FUNCTION_BLOCK PUBLIC RejectStation
VAR_INPUT
END_VAR
VAR_OUTPUT
END_VAR
VAR
	xTrigger :BOOL := FALSE; // triggers processing
	State : eRejectStaState := eRejectStaState.eUnknown;
	NextState : eRejectStaState := eRejectStaState.eUnknown;
	ErrorReturnState : eRejectStaState := eRejectStaState.eUnknown;
	bFirst : BOOL := TRUE;
	VUT : BYTE; //VehicleID Under Station
	DwellTimer : TON;
	StateTimer : TON;
END_VAR

IF (GVL_IO.MachineEStopped) THEN 
	State := eRejectStaState.eUnknown;
	NextState := eRejectStaState.eUnknown;
	Status.RejectStatusMsg:= 'RejectSta Unknown, Check AIR, E-STOP and Hit Start';
END_IF

CASE State OF
eRejectStaState.eUnknown:
	Status.RejectStatusMsg:= 'RejectSta Unknown, Check AIR, E-STOP and Hit Start';
    IF (GVL_IO.MC_XStartPB AND GVL_IO.MC_XAirPressureOK AND GVL_IO.MC_NotEStopped) THEN // wait for start button when powered up or PLC program restarted
		NextState := eRejectStaState.eInit;	   
	END_IF
    

eRejectStaState.eInit:
    Act_KnockPartOFF();
	Act_FreePalletHoldDown();
	ResetDwellTimer();
	NextState := eRejectStaState.eHoming;
	

eRejectStaState.eHoming:
	IF (IsPalletHoldDownFree()) THEN 
         NextState := eRejectStaState.eReady;
	  END_IF
     DwellTimer(IN:=TRUE, PT:= T#10S);
     IF (DwellTimer.Q) THEN
		 ResetDwellTimer();
		 ErrorReturnState:= eRejectStaState.eInit;
		 NextState := eRejectStaState.eError;		 
	 END_IF	

eRejectStaState.eReady:
	IF (xTrigger) THEN
		NextState := eRejectStaState.eSendPalletHoldDownExtend;		
		ResetDwellTimer();
	END_IF

eRejectStaState.eSendPalletHoldDownExtend:
	Act_EngagePalletHoldDown();
	ResetDwellTimer();
	NextState := eRejectStaState.eCheckPalletHoldDownExtended;
	
eRejectStaState.eCheckPalletHoldDownExtended:
   DwellTimer(IN:=TRUE, PT:= T#10S);	
   IF (IsPalletHoldDownEngaged()) THEN
        ResetDwellTimer();	   
		IF(GVL_IO.RJ_XPartPresent OR TRUE) THEN         //added Turnkey shop sensor not adjusted
			NextState := eRejectStaState.eKnockOffPart;
			ResetDwellTimer();
        ELSE
			NextState := eRejectStaState.ePalletHoldDownRelease;	
		END_IF        
   END_IF      
   IF (DwellTimer.Q) THEN
		 ResetDwellTimer();
		 ErrorReturnState:= eRejectStaState.eSendPalletHoldDownExtend;
		 NextState := eRejectStaState.eError;		 
	END_IF
  
eRejectStaState.eKnockoffPart:
	Act_KnockPartON();
	UpdateLotData();
	UpdatePartData();
    DwellTimer(IN:=TRUE, PT:= T#250MS);
    IF (DwellTimer.Q) THEN 
		NextState := eRejectStaState.eCheckPartKnockedOff;
		ResetDwellTimer();
	END_IF;

eRejectStaState.eCheckPartKnockedOff:
   IF (NOT(GVL_IO.RJ_XPartPresent) ) THEN   /// until Bonnie can ajust sensor
	   NextState := eRejectStaState.ePalletHoldDownRelease;
	   DwellTimer(IN:=FALSE);
	   StateTimer(IN:=FALSE);
   END_IF
   DwellTimer(IN:= TRUE, PT:= T#10S);
   IF (DwellTimer.Q) THEN
	   ResetDwellTimer();
	   ErrorReturnState:= eRejectStaState.eCheckPartKnockedOff;
	   Status.RejectStatusMsg:= 'Reject Remove Part then Hit START';
   	   NextState := eRejectStaState.eError;	
   END_IF   

eRejectStaState.ePalletHoldDownRelease:
    Act_KnockPartOFF();
	Act_FreePalletHoldDown();
    ResetDwellTimer();	
	NextState := eRejectStaState.ePalletHoldDownReleased;

eRejectStaState.ePalletHoldDownReleased:	
	IF (IsPalletHoldDownFree()) THEN         
	    NextState := eRejectStaState.eDepart;
    END_IF
	
   DwellTimer(IN:= TRUE, PT:= T#10S);
   IF (DwellTimer.Q) THEN
	   ResetDwellTimer();
	   ErrorReturnState:= eRejectStaState.ePalletHoldDownRelease;	   
   	   NextState := eRejectStaState.eError;	
   END_IF  
	
	
eRejectStaState.eDepart:
    Stations.fbRoutePlanner.M_NotifyVehStaCmpl(StationIndex:= MM_CONST.REJECT_ULOAD_STA, VehicleID := VUT);
	xTrigger := FALSE;
	IF (Stations.fbCycleControl.StopRequested) THEN
		NextState := eRejectStaState.eStopActive;
	ELSE 
		NextState := eRejectStaState.eReady;
    END_IF
	
eRejectStaState.eStopActive:
	IF (NOT Stations.fbCycleControl.StopRequested) THEN
		NextState := eRejectStaState.eReady;
    END_IF
	

eRejectStaState.eError:
	IF (GVL_IO.MC_XStartPB) THEN
		NextState := ErrorReturnState;
		ErrorReturnState := eRejectStaState.eUnknown;
	END_IF

END_CASE

IF (State <> NextState) THEN
	bFirst := TRUE;
	StateTimer(IN:=FALSE);
ELSE
	bFirst := FALSE;
END_IF

State := NextState;
AssignStationStatusForHMI();

ACTION Act_EngagePalletHoldDown:
GVL_IO.RJ_YPalletHoldDownExtend_Home  := FALSE;
GVL_IO.RJ_YPalletHoldDownRetract_Engage := TRUE;
END_ACTION

ACTION Act_FreePalletHoldDown:
GVL_IO.RJ_YPalletHoldDownExtend_Home := TRUE;
GVL_IO.RJ_YPalletHoldDownRetract_Engage := FALSE;
END_ACTION

ACTION Act_KnockPartOFF:
	GVL_IO.RJ_YRejectPushExtend := FALSE;
	GVL_IO.RJ_YRejectPushRetract := TRUE;
END_ACTION

ACTION Act_KnockPartON:
	GVL_IO.RJ_YRejectPushExtend := TRUE;
	GVL_IO.RJ_YRejectPushRetract := FALSE;
END_ACTION

METHOD PUBLIC AssignStationStatusForHMI : BOOL
VAR_INPUT
END_VAR
Status.StationsState[MM_CONST.REJECT_ULOAD_STA_HMI_STATE] := State;
IF (NOT LotsData.Lot.RejectUnloadEnabled) THEN
	Status.StationStauts[MM_CONST.REJECT_ULOAD_STA_HMI_STATE] := OverallStationStatus.eDisabled;
ELSE 
	CASE State OF 
	
	eRejectStaState.eUnknown,eRejectStaState.eError:
		Status.StationStauts[MM_CONST.REJECT_ULOAD_STA_HMI_STATE] := OverallStationStatus.eError;
		
    eRejectStaState.eInit,
	eRejectStaState.eHoming:
	    Status.StationStauts[MM_CONST.REJECT_ULOAD_STA_HMI_STATE] := OverallStationStatus.eHoming;
	
	eRejectStaState.eReady,eRejectStaState.eWaitForVehicleTrigger:
	     Status.StationStauts[MM_CONST.REJECT_ULOAD_STA_HMI_STATE] := OverallStationStatus.eWaitingForParts;
		 
	eRejectStaState.eDwell,
	eRejectStaState.eSendPalletHoldDownExtend,
	eRejectStaState.eCheckPalletHoldDownExtended,
	eRejectStaState.ePalletReleaseExtend,
	eRejectStaState.ePalletReleaseExtended,
	eRejectStaState.eKnockoffPart,
	eRejectStaState.eKnockoffExtended,
	eRejectStaState.eCheckPartKnockedOff,
	eRejectStaState.ePalletHoldDownRelease,
	eRejectStaState.ePalletHoldDownReleased:
	    Status.StationStauts[MM_CONST.REJECT_ULOAD_STA_HMI_STATE] := OverallStationStatus.eRunning;
	
	eRejectStaState.eStopActive:
	    Status.StationStauts[MM_CONST.REJECT_ULOAD_STA_HMI_STATE] := OverallStationStatus.eCycleStop;
    	
	
    ELSE;	
	END_CASE
END_IF
END_METHOD

METHOD PUBLIC ClearVehicleTrigger : BOOL
VAR_INPUT
END_VAR
xTrigger := FALSE;
END_METHOD

METHOD PUBLIC IsFaulted : BOOL
VAR_INPUT
END_VAR
IsFaulted := (State = eRejectStaState.eUnknown OR State = eRejectStaState.eError);
END_METHOD

METHOD PUBLIC IsPalletHoldDownEngaged : BOOL
VAR_INPUT
END_VAR
IsPalletHoldDownEngaged := (GVL_IO.RJ_XPalletHoldDownRetracted_Engaged AND NOT GVL_IO.RJ_XPalletHoldDownExtended_Home);
IF (NOT IsPalletHoldDownEngaged) THEN
	Status.RejectStatusMsg:= 'Reject: Check Pallet Hold Down Sensors and then hit START';
END_IF
END_METHOD

METHOD PUBLIC IsPalletHoldDownFree : BOOL
VAR_INPUT
END_VAR
IsPalletHoldDownFree := (NOT GVL_IO.RJ_XPalletHoldDownRetracted_Engaged AND GVL_IO.RJ_XPalletHoldDownExtended_Home);
IF (NOT IsPalletHoldDownFree) THEN
	Status.RejectStatusMsg:= 'Reject: Check Pallet Hold Down Sensors and then hit START';
END_IF
END_METHOD

PROPERTY PUBLIC Ready : BOOL
GET
Ready := (State = eRejectStaState.eReady);
END_GET
END_PROPERTY

ACTION ResetDwellTimer:
DwellTimer(IN:=FALSE);
END_ACTION

METHOD PUBLIC ResetState : BOOL
VAR_INPUT
END_VAR
State := eRejectStaState.eUnknown;
NextState := eRejectStaState.eUnknown;
END_METHOD

PROPERTY PUBLIC Trigger : BOOL
SET
xTrigger := Trigger;
END_SET
END_PROPERTY

METHOD PUBLIC UpdateLotData : BOOL
VAR_INPUT
END_VAR
IF (PartsData.Status[VUT].OverallStatus <> ePartStatus.eEmpty) THEN
	LotsData.Lot.CavityCounts[PartsData.Status[VUT].CavityNumber].BadCount := LotsData.Lot.CavityCounts[PartsData.Status[VUT].CavityNumber].BadCount +1;
	LotsData.Lot.CavityCounts[PartsData.Status[VUT].CavityNumber].TotalCount := LotsData.Lot.CavityCounts[PartsData.Status[VUT].CavityNumber].TotalCount + 1;
END_IF
END_METHOD

METHOD PUBLIC UpdatePartData : BOOL
VAR_INPUT
END_VAR
PartsData.Status[VUT].RejectUnloadTime := SYSTEMTIME_TO_STRING(Logging.fbCurrTime.systemTime);
IF (PartsData.Status[VUT].OverallStatus <> ePartStatus.eEmpty) THEN
	IF (P_TextModeWrite.CurrWriteStep = 0) THEN (* if resource not ready, we will skip this part*)
    P_TextModeWrite.VehicleID := VUT;
	P_TextModeWrite.WriteData := TRUE;
	END_IF 
END_IF
PartsData.Status[VUT].OverallStatus := ePartStatus.eEmpty;

// we will write data to CSV file over here
END_METHOD

PROPERTY PUBLIC VehicleUnderTest : BYTE
GET
VehicleUnderTest := VUT;
END_GET
SET
VUT := VehicleUnderTest;
END_SET
END_PROPERTY

END_FUNCTION_BLOCK

(* stored: Version 1.1.0.1, ProductVersion 3.1.4022.6
   POU RejectStation: Id {1c7d3c10-2e05-4827-bb38-6a50101bbab4}, SpecialFunc None
   Action Act_EngagePalletHoldDown: Id {3f30117c-5e6e-48a8-b3a1-5e4bdf95c3b8}
   Action Act_FreePalletHoldDown: Id {31d36249-0615-4b2f-8d93-d911987274cd}
   Action Act_KnockPartOFF: Id {0dd1b6cc-028c-4568-86b1-43e1daf5b4c5}
   Action Act_KnockPartON: Id {bbe591a0-cc44-44b8-88ed-b7df52180766}
   Method AssignStationStatusForHMI: Id {9daeb57e-5015-4a77-b83a-e539e06cc06a}
   Method ClearVehicleTrigger: Id {976b5edd-4b06-4989-a8bc-6ca4b3cd4f57}
   Method IsFaulted: Id {d3043999-8417-49a5-b283-6c2328820a8c}
   Method IsPalletHoldDownEngaged: Id {a11e39c7-24b4-48ba-8798-808616fedafe}
   Method IsPalletHoldDownFree: Id {63e2664c-f6cb-45b3-9777-3cb53c2f81e3}
   Property Ready: Id {e36dc20c-e8de-419a-9137-4af11dd3af4e}
   Get Get: Id {35b042ee-ce62-4e99-b7a2-97e5b91ab954}
   Action ResetDwellTimer: Id {ebefa544-ef12-4966-9806-2e0b5908407f}
   Method ResetState: Id {9f7b9e0a-4ac5-4c94-9069-f97240cf99ca}
   Property Trigger: Id {47817a75-f5a0-4907-8635-da34a5b57ff9}
   Set Set: Id {5ef6f9b5-5847-4fc5-ac2e-197e7eb892a4}
   Method UpdateLotData: Id {c1f12ee8-8147-4650-9883-b6863bf398be}
   Method UpdatePartData: Id {9d30b08e-a5ef-452c-8b03-271af7fbf7ce}
   Property VehicleUnderTest: Id {b50b124c-8e38-4d9a-a197-9c352deb6071}
   Get Get: Id {de905004-ffa8-4240-8f99-7740d1f80dc6}
   Set Set: Id {7e6b83d6-a21a-48cd-a2cd-76093cb1c9f7} *)
